// TIA Portal V19 export
FUNCTION_BLOCK "LAF_PlcDiag"   // FB22, LAD
TITLE = LAF_PlcDiag / SPS Geraete Status
AUTHOR : Siemens Digital Industries
FAMILY : LAF
VERSION : 1.2
// The block reads the identification and maintenance data (I&M data) as well as the network addresses from the PLC and provides the information in the screen “Settings – PLC identification“. The screen is accessible in the setting screen.  
// 
// **PLC Data types**  
// * LAF_typePlcDiag  
// 
// **WinCC Screen**  
// ![Image](LAF_PlcDiag/en/image1.PNG)  
// 
// ---
// 
// **Block call example**  
// ![Image](LAF_PlcDiag/en/image5.PNG)  
// 
// ---
// 
// **Calling interface**  
// The block will be called once only in the cyclic program. The call takes place in the software unit CentralFunctions -> 05_Diagnostics -> [CallDiagnostic](../Functions/CallDiagnostic.htm)  
// 
// **Internally used “Extended instructions / blocks“**  
// GET_IM_DATA, RDREC, S_CONV, MOVE_BLK_VARIANT  
// 
// **Parameters**  
// This block is provided with “pre-defined actual parameters” for structured data types, user constants, system constants etc. Therefor these parameters have to be modified only slightly or not at all, if the symbols of DBs, user constants, and system constants have not been changed.  
// In the case of LAF_PlcDiag you only have to write the correct information on the input parameter localProfinetInterface.
// 
// **Get parameter information:**..
// **localCommon**  
// ![Image](LAF_PlcDiag/en/image2.PNG)  
// 
// ---
// 
// **localProfinetInterface**  
// ![Image](LAF_PlcDiag/en/image3.PNG)
// Der Baustein liest die Identification und Maintenance Daten (I&M-Daten), sowie die Netzwerkadressen der CPU aus und stellt diese in dem Bild „SYSTEM_SETTINGS“ zur Verfügung. Das Bild ist erreichbar über den Button „System“ (aus jedem Bild, rechts unten).  
// 
// **PLC-Datentypen**  
//  LSicar_typePlcDiag  
//  
// **WinCC-Bild**  
// 
// ![Image](LSicar_typePlcDiag/de/image1.PNG)  
// 
// **Beispielaufruf**  
// Abbildung in Kontaktplan (KOP), ohne Parameterbeschaltung. D:\Software\Symbols_Icons\BMPs-JPGs-PNGs\Verschiedene\symb_user_goto_transparent.pngEin lauffähiger Programm-Aufruf hierzu ist im „SICAR-StartUp“-Projekt enthalten, incl. der notwendigen HMI-Variablen zur Darstellung der der Werte auf dem HMI.  
// 
// **Aufrufschnittstelle**  
// Der Baustein wird einmalig im zyklischen Programm aufgerufen.  
// 
// **Intern verwendete „Erweiterte Anweisungen / Bausteine“**  
// GET_IM_DATA, RDREC, S_CONV, MOVE_BLK_VARIANT 
// 
// **Parameter**  
// Der Baustein ist mit "Vordefinierten Aktualparametern" versehen für Strukturvariablen, Anwender- und Systemkonstanten etc., die dadurch nicht oder nur geringfügig angepasst werden müssen, vorausgesetzt die Symbolischen Namen von DBs, Anwender-/Systemkonstanten etc. wurden nicht geändert. Die Anpassungen sind notwendig beim Index [i], z.B. für den BA-Bereich oder die HMI-/Panelnummer.  
// * Der Index ist vorbesetzt mit dem Wert [0]. Damit wird auf den Index 0 (Dummy) verwiesen. Sofern der Baustein-Parameter nicht benötigt wird, sind keine Anpassungen notwendig, andernfalls muss der Indexwert angepasst werden. 
// oder  
// * Der Index ist vorbesetzt mit [???]. Dies führt dazu, dass der Aktualparameter beim Bausteinaufruf rot markiert wird; um darauf aufmerksam zu machen, dass der Indexwert des Aktualparameters angepasst werden muss!
// stored: Access Published, IsIECCheckEnabled true, MemoryReserve 100, SetENOAutomatically true
   VAR_INPUT
      localCommon { ExternalAccessible := 'False'; ExternalVisible := 'False'; ExternalWritable := 'False'} : HW_SUBMODULE;   // Systemkonstante: Local~PROFINET_IO-System / System constant: Local~Common
      localProfinetInterface { ExternalAccessible := 'False'; ExternalVisible := 'False'; ExternalWritable := 'False'} : HW_INTERFACE;   // Systemkonatante: Local~PROFINET-Interface_... / System constant: Local~PROFINET-Interface_...
      firstCycle { ExternalAccessible := 'False'; ExternalVisible := 'False'; ExternalWritable := 'False'} : Bool;   // SystemFlag: FirstCycle / System Flag: FirstCycle
   END_VAR
   VAR_IN_OUT
      diagDataHmi : "LAF_typePlcDiag";   // PLC-Diagnostic Data
   END_VAR
   VAR
      statLocalCommon { ExternalAccessible := 'False'; ExternalVisible := 'False'; ExternalWritable := 'False'} : HW_SUBMODULE;   // HW submodul
      statLocProfinetInterface { ExternalAccessible := 'False'; ExternalVisible := 'False'; ExternalWritable := 'False'} : HW_INTERFACE;   // HW interface
      instGetImData0 { ExternalAccessible := 'False'; ExternalVisible := 'False'; ExternalWritable := 'False'} : Get_IM_Data;   // I&M 0-Daten
      statGetImData0ErrorSaved { ExternalAccessible := 'False'; ExternalVisible := 'False'; ExternalWritable := 'False'} : Word;   // I&M 0-Daten
      instGetImData1 { ExternalAccessible := 'False'; ExternalVisible := 'False'; ExternalWritable := 'False'} : Get_IM_Data;   // I&M 1-Daten
      statGetImData1ErrorSaved { ExternalAccessible := 'False'; ExternalVisible := 'False'; ExternalWritable := 'False'} : Word;   // I&M 1-Daten
      instGetImData2 { ExternalAccessible := 'False'; ExternalVisible := 'False'; ExternalWritable := 'False'} : Get_IM_Data;   // I&M 2-Daten
      statGetImData2ErrorSaved { ExternalAccessible := 'False'; ExternalVisible := 'False'; ExternalWritable := 'False'} : Word;   // I&M 2-Daten
      instGetImData3 { ExternalAccessible := 'False'; ExternalVisible := 'False'; ExternalWritable := 'False'} : Get_IM_Data;   // I&M 3-Daten
      statGetImData3ErroSaved { ExternalAccessible := 'False'; ExternalVisible := 'False'; ExternalWritable := 'False'} : Word;   // I&M 3-Daten
      instReadRecord { ExternalAccessible := 'False'; ExternalVisible := 'False'; ExternalWritable := 'False'} : RDREC;   // RDREC
      statReadRecordResult { ExternalAccessible := 'False'; ExternalVisible := 'False'; ExternalWritable := 'False'} : Array[0..199] of Byte;   // RDREC-Record
      statStartNetAddresses { ExternalAccessible := 'False'; ExternalVisible := 'False'; ExternalWritable := 'False'} : USInt;   // Anfang der Netzadressesn (MAC, IP, Subnet, ...) / Start of net adresses (MAC, IP, Subnet, ...)
      statIm1PlDesiLocIdLen { ExternalAccessible := 'False'; ExternalVisible := 'False'; ExternalWritable := 'False'} : Int;   // Länge/Anzahl Zeichen von String "IuM_1_PlantDesign_LocIdent" / Lenght/Number of signs of string "IuM_1_PlantDesign_LocIdent"
      statRisEdgeReadAll { ExternalAccessible := 'False'; ExternalVisible := 'False'; ExternalWritable := 'False'} : Bool;   // Rising edge read all / Steigende Flanke read all
      statPosPulseReadAll { ExternalAccessible := 'False'; ExternalVisible := 'False'; ExternalWritable := 'False'} : Bool;   // Pos pulse read all / Pos. Impuls read all
      statErrorText { ExternalAccessible := 'False'; ExternalVisible := 'False'; ExternalWritable := 'False'} : String[#LENGTH_ERROR_TEXT] := STRING#'Error - Not readable data';   // Error text / Fehlertext
   END_VAR
   VAR_TEMP
      tempNetAddress : USInt;   // Netzadresse / Net address
      tempReadRecordResult6 : USInt;   // Type conversion / Typ Konvertierung
   END_VAR
   VAR CONSTANT
      VALUE_2 : USInt := 2;   // Konstante 2 / Const 2
      VALUE_4 : USInt := 4;   // 4Byte-1DW / 4 byte-1DW
      INDEX_ADDRESS_1ST_SIGN : USInt := 6;   // Indexadresse 1.Zeichen / Index address
      LENGTH_ERROR_TEXT : DInt := 30;   // Length error text / Zeichenlänge Fehlertext
   END_VAR
   VAR_TEMP   // added for the SCL form of the ladder/FBD networks
      _w1 : Bool;
   END_VAR
BEGIN

REGION Network 1: Header Info / Änderungshistorie
   // SIEMENS AG / (c)Copyright 2024
   // ------------------------------------------------------------------------------
   // Title:            LAF_InterfaceSignalsBool
   // Comment/Function: The block reads the identification and maintenance data (I&M data) as well as the network addresses from the PLC and provides the information in the screen “Settings – PLC identification“. 
   // Library/Family:  Library of Automation Framework
   // Author:               Siemens Digital Industry
   // Tested with:      S7-PLCSIM Advanced 6.0
   // Engineering:     TIA Portal V19
   // Restrictions:      ---
   // Requirements:  ---
   // ------------------------------------------------------------------------------
   // Change log table:
   // Version | Date | Expert in charge | Changes applied
   // -------|---------|-------------|--------------------------------------------
   // 01.02.00 | 30.09.2024 | SIMATIC Systems Support | First released version
   // Die Änderungshistorie wird nur in englischer Editiersprache geführt.
END_REGION

REGION Network 2: Description / Beschreibung
   // **Operation mode Automatic / Manual**  
   // The block is not assigned to any operation mode.  
   // 
   // **Alarms**  
   // The block does not generate alarms.  
   // 
   // #### PLC Data types 
   // * [LAF_typePlcDiag](../Library%20Types/LAF_typePlcDiag.htm)  
   // 
   // #### WinCC-Screen objects  
   // 
   // **WinCC Screen**  
   // The screen is located in the project in HMI part under “Screens” -> “11_Settings”.  
   // It consists of several WinCC objects and contains the shown below information.  
   // The Identification and Maintenance Data as well as the CPU net addresses are read once after a CPU warm start and displayed in the shown screen.  
   // ![Image](LAF_PlcDiag/en/image4.PNG)  
   // 
   // 
   // #### Further information 
   // 
   // #### Update info 
   // 
   // #### Further documentation
   // **Betriebsart Automatik / Hand**  
   // Der Baustein ist keiner Betriebsart / Betriebsartenbereich zugeordnet.  
   // 
   // **Alarme**  
   // Der Baustein generiert keine Alarme.  
   // 
   // #### PLC-Datentypen 
   // Der PLC-Datentyp „_typePlcDiag“ enthält alle Informationen, die in der Visualisierung angezeigt werden.  
   // 
   // #### WinCC-Bildobjekte 
   // **WinCC-Bild**  
   // Das Bild befindet sich im Projekt im HMI-Teil unter „Bilder“. Es ist erstellt aus mehreren einzelnen WinCC-Objekten und enthält die dargestellten Informationen.  
   // 
   // ![Image](LSicar_typePlcDiag/de/image2.PNG) 
   // 
   // 
   // #### Weitere Hinweise
   // 
   // #### Updateinfo 
   // 
   // #### Weitere Dokumente
END_REGION

REGION Network 3: Preset values after restart / Werte vorbesetzen nach Neustart
   // Initialization of the values / Initialisieren der  Werte
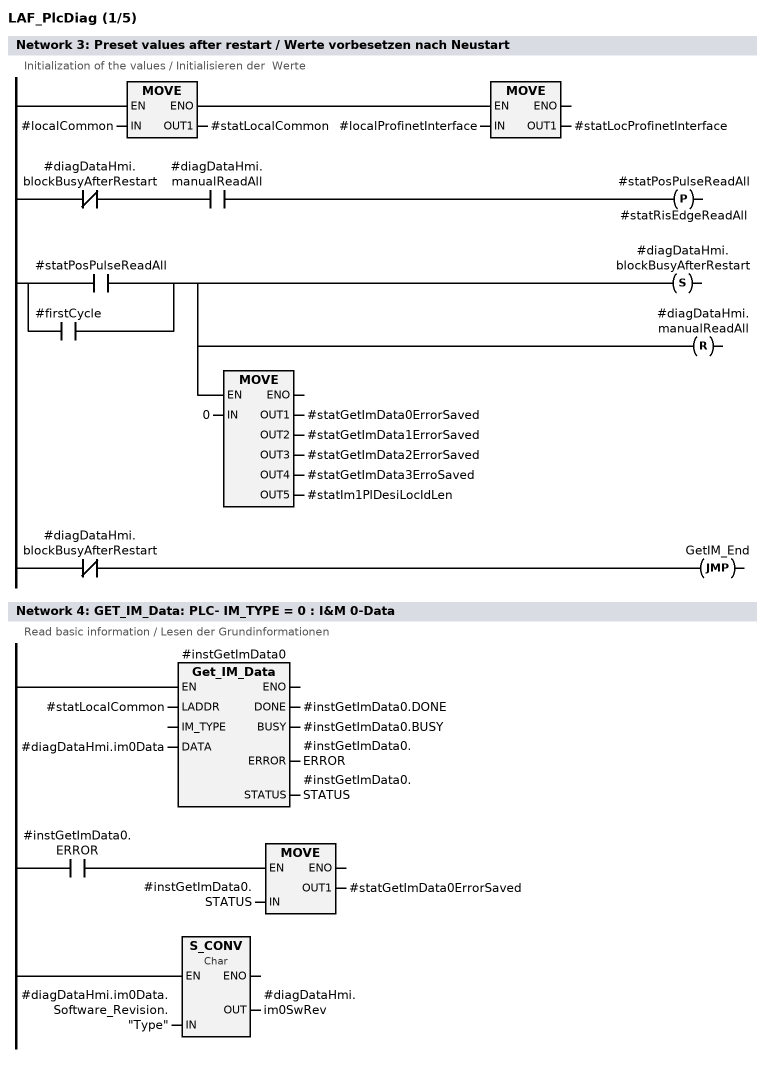
   #statLocalCommon := #localCommon;
   #statLocProfinetInterface := #localProfinetInterface;
   #_w1 := NOT #diagDataHmi.blockBusyAfterRestart AND #diagDataHmi.manualReadAll;
   #statPosPulseReadAll := #_w1 AND NOT #statRisEdgeReadAll;   // rising edge
   #statRisEdgeReadAll := #_w1;
   IF #statPosPulseReadAll OR #firstCycle THEN
       #diagDataHmi.blockBusyAfterRestart := TRUE;
       #diagDataHmi.manualReadAll := FALSE;
       #statGetImData0ErrorSaved := 0;
       #statGetImData1ErrorSaved := 0;
       #statGetImData2ErrorSaved := 0;
       #statGetImData3ErroSaved := 0;
       #statIm1PlDesiLocIdLen := 0;
   END_IF;
   IF NOT #diagDataHmi.blockBusyAfterRestart THEN GOTO GetIM_End; END_IF;
END_REGION

REGION Network 4: GET_IM_Data: PLC- IM_TYPE = 0 : I&M 0-Data
   // Read basic information / Lesen der Grundinformationen
   RUNG wire#powerrail
      #instGetImData0.Get_IM_Data(LADDR := #statLocalCommon, IM_TYPE :=, DATA := #diagDataHmi.im0Data, DONE => #instGetImData0.DONE, BUSY => #instGetImData0.BUSY, ERROR => #instGetImData0.ERROR, STATUS => #instGetImData0.STATUS)
   END_RUNG
   RUNG wire#powerrail
      Contact( #instGetImData0.ERROR )
      Move(in := #instGetImData0.STATUS, out1 => #statGetImData0ErrorSaved)
   END_RUNG
   RUNG wire#powerrail
      { S7_Templates := "[src_type := Char, dest_type := String]" } S_CONV(IN := #diagDataHmi.im0Data.Software_Revision."Type", OUT => #diagDataHmi.im0SwRev)
   END_RUNG
   // the same network as SCL:
   #instGetImData0(LADDR := #statLocalCommon,   // Get_IM_Data
                   DATA := #diagDataHmi.im0Data,
                   DONE => #instGetImData0.DONE,
                   BUSY => #instGetImData0.BUSY,
                   ERROR => #instGetImData0.ERROR,
                   STATUS => #instGetImData0.STATUS);
   IF #instGetImData0.ERROR THEN #statGetImData0ErrorSaved := #instGetImData0.STATUS; END_IF;
   S_CONV(IN := #diagDataHmi.im0Data.Software_Revision."Type", OUT => #diagDataHmi.im0SwRev);
END_REGION

REGION Network 5: GET_IM_Data: PLC- IM_TYPE = 11: I&M 1-Data
   // Read functional description an designation of the PLC / Lesen der Functionsbeschreibung und Bezeichnung der SPS
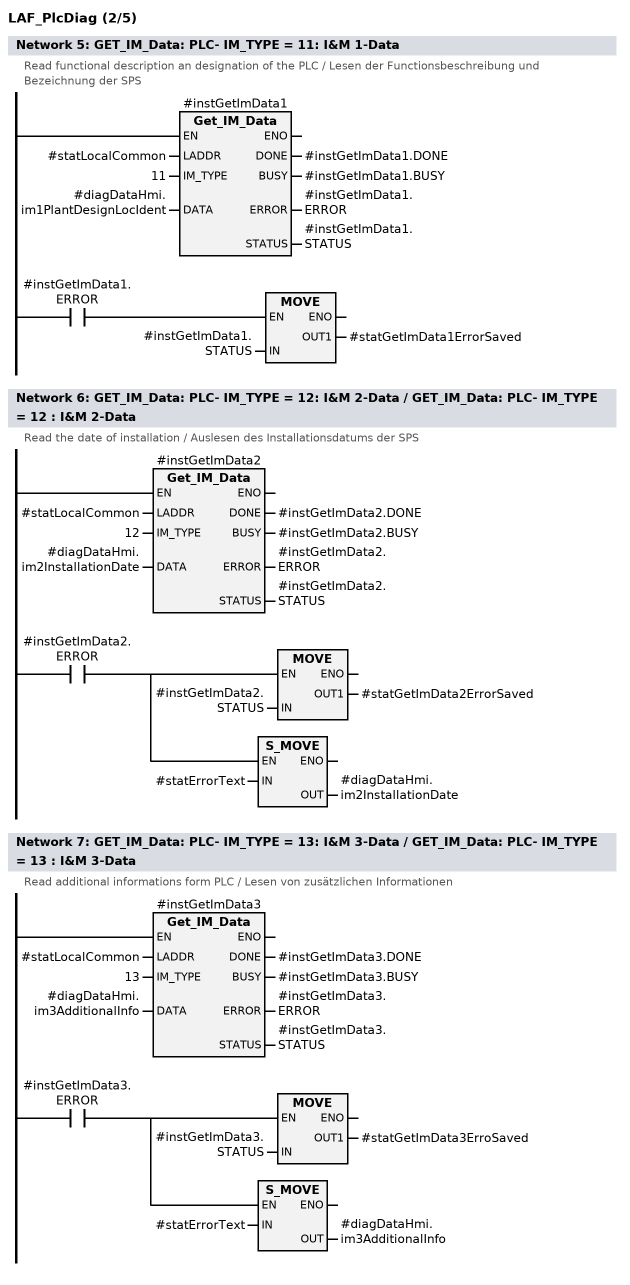
   RUNG wire#powerrail
      #instGetImData1.Get_IM_Data(LADDR := #statLocalCommon, IM_TYPE := 11, DATA := #diagDataHmi.im1PlantDesignLocIdent, DONE => #instGetImData1.DONE, BUSY => #instGetImData1.BUSY, ERROR => #instGetImData1.ERROR, STATUS => #instGetImData1.STATUS)
   END_RUNG
   RUNG wire#powerrail
      Contact( #instGetImData1.ERROR )
      Move(in := #instGetImData1.STATUS, out1 => #statGetImData1ErrorSaved)
   END_RUNG
   // the same network as SCL:
   #instGetImData1(LADDR := #statLocalCommon,   // Get_IM_Data
                   IM_TYPE := 11,
                   DATA := #diagDataHmi.im1PlantDesignLocIdent,
                   DONE => #instGetImData1.DONE,
                   BUSY => #instGetImData1.BUSY,
                   ERROR => #instGetImData1.ERROR,
                   STATUS => #instGetImData1.STATUS);
   IF #instGetImData1.ERROR THEN #statGetImData1ErrorSaved := #instGetImData1.STATUS; END_IF;
END_REGION

REGION Network 6: GET_IM_Data: PLC- IM_TYPE = 12: I&M 2-Data / GET_IM_Data: PLC- IM_TYPE = 12 : I&M 2-Data
   // Read the date of installation / Auslesen des Installationsdatums der SPS
   RUNG wire#powerrail
      #instGetImData2.Get_IM_Data(LADDR := #statLocalCommon, IM_TYPE := 12, DATA := #diagDataHmi.im2InstallationDate, DONE => #instGetImData2.DONE, BUSY => #instGetImData2.BUSY, ERROR => #instGetImData2.ERROR, STATUS => #instGetImData2.STATUS)
   END_RUNG
   RUNG wire#powerrail
      Contact( #instGetImData2.ERROR )
      wire#w1
      Move(in := #instGetImData2.STATUS, out1 => #statGetImData2ErrorSaved)
   END_RUNG
   RUNG wire#w1
      S_Move(in := #statErrorText, out => #diagDataHmi.im2InstallationDate)
   END_RUNG
   // the same network as SCL:
   #instGetImData2(LADDR := #statLocalCommon,   // Get_IM_Data
                   IM_TYPE := 12,
                   DATA := #diagDataHmi.im2InstallationDate,
                   DONE => #instGetImData2.DONE,
                   BUSY => #instGetImData2.BUSY,
                   ERROR => #instGetImData2.ERROR,
                   STATUS => #instGetImData2.STATUS);
   IF #instGetImData2.ERROR THEN
       #statGetImData2ErrorSaved := #instGetImData2.STATUS;
       #diagDataHmi.im2InstallationDate := #statErrorText;
   END_IF;
END_REGION

REGION Network 7: GET_IM_Data: PLC- IM_TYPE = 13: I&M 3-Data / GET_IM_Data: PLC- IM_TYPE = 13 : I&M 3-Data
   // Read additional informations form PLC / Lesen von zusätzlichen Informationen
   RUNG wire#powerrail
      #instGetImData3.Get_IM_Data(LADDR := #statLocalCommon, IM_TYPE := 13, DATA := #diagDataHmi.im3AdditionalInfo, DONE => #instGetImData3.DONE, BUSY => #instGetImData3.BUSY, ERROR => #instGetImData3.ERROR, STATUS => #instGetImData3.STATUS)
   END_RUNG
   RUNG wire#powerrail
      Contact( #instGetImData3.ERROR )
      wire#w1
      Move(in := #instGetImData3.STATUS, out1 => #statGetImData3ErroSaved)
   END_RUNG
   RUNG wire#w1
      S_Move(in := #statErrorText, out => #diagDataHmi.im3AdditionalInfo)
   END_RUNG
   // the same network as SCL:
   #instGetImData3(LADDR := #statLocalCommon,   // Get_IM_Data
                   IM_TYPE := 13,
                   DATA := #diagDataHmi.im3AdditionalInfo,
                   DONE => #instGetImData3.DONE,
                   BUSY => #instGetImData3.BUSY,
                   ERROR => #instGetImData3.ERROR,
                   STATUS => #instGetImData3.STATUS);
   IF #instGetImData3.ERROR THEN
       #statGetImData3ErroSaved := #instGetImData3.STATUS;
       #diagDataHmi.im3AdditionalInfo := #statErrorText;
   END_IF;
END_REGION

REGION Network 8: Read IP adress / Lesen der IP Adresse
   // Once only read RDREC (IP-Adresse): after PLC-restart or manual read from HMI / Einmaliges Lesen RDREC: nach SPS - Neustart oder manueller Anstoss vom HMI
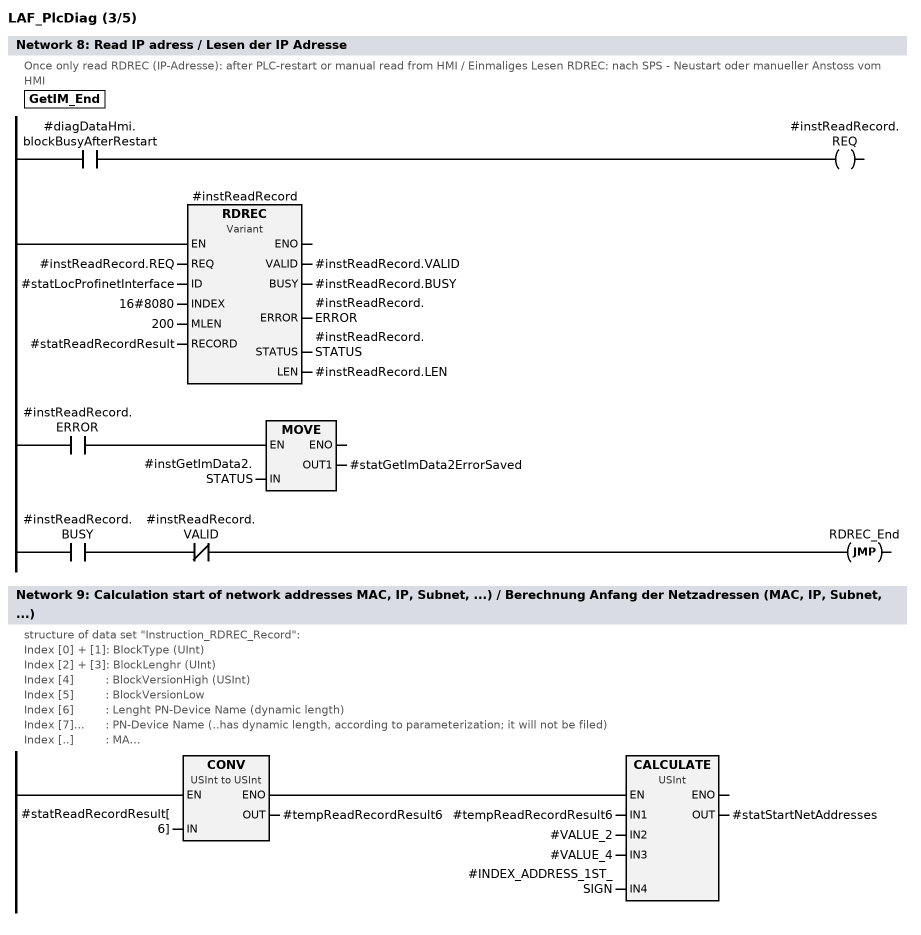
   Label( GetIM_End )
   RUNG wire#powerrail
      Contact( #diagDataHmi.blockBusyAfterRestart )
      Coil( #instReadRecord.REQ )
   END_RUNG
   RUNG wire#powerrail
      { S7_Templates := "[ptr_type := Variant, id_type := HW_IO, index_type := DInt, len_type := UInt]" } #instReadRecord.RDREC(REQ := #instReadRecord.REQ, ID := #statLocProfinetInterface, INDEX := 16#8080, MLEN := 200, RECORD := #statReadRecordResult, VALID => #instReadRecord.VALID, BUSY => #instReadRecord.BUSY, ERROR => #instReadRecord.ERROR, STATUS => #instReadRecord.STATUS, LEN => #instReadRecord.LEN)
   END_RUNG
   RUNG wire#powerrail
      Contact( #instReadRecord.ERROR )
      Move(in := #instGetImData2.STATUS, out1 => #statGetImData2ErrorSaved)
   END_RUNG
   RUNG wire#powerrail
      Contact( #instReadRecord.BUSY )
      I_Contact( #instReadRecord.VALID )
      JumpCoil( RDREC_End )
   END_RUNG
   // the same network as SCL:
   GetIM_End:
   #instReadRecord.REQ := #diagDataHmi.blockBusyAfterRestart;
   #instReadRecord(REQ := #instReadRecord.REQ,   // RDREC
                   ID := #statLocProfinetInterface,
                   INDEX := 16#8080,
                   MLEN := 200,
                   RECORD := #statReadRecordResult,
                   VALID => #instReadRecord.VALID,
                   BUSY => #instReadRecord.BUSY,
                   ERROR => #instReadRecord.ERROR,
                   STATUS => #instReadRecord.STATUS,
                   LEN => #instReadRecord.LEN);
   IF #instReadRecord.ERROR THEN #statGetImData2ErrorSaved := #instGetImData2.STATUS; END_IF;
   IF #instReadRecord.BUSY AND NOT #instReadRecord.VALID THEN GOTO RDREC_End; END_IF;
END_REGION

REGION Network 9: Calculation start of network addresses MAC, IP, Subnet, ...) / Berechnung Anfang der Netzadressen (MAC, IP, Subnet, ...)
   // structure of data set "Instruction_RDREC_Record":
   // Index [0] + [1]: BlockType (UInt)
   // Index [2] + [3]: BlockLenghr (UInt)
   // Index [4]         : BlockVersionHigh (USInt)
   // Index [5]         : BlockVersionLow
   // Index [6]         : Lenght PN-Device Name (dynamic length)
   // Index [7]...      : PN-Device Name (..has dynamic length, according to parameterization; it will not be filed)
   // Index [..]         : MAC
   // Index [..]         : IP
   // Index [..]         : SubnetMask
   // Index [..]         : Standard Gateway (is not filed)
   // Aufbau des Datensatzes "Instruction_RDREC_Record":
   // Index [0] + [1]: BlockType (UInt)
   // Index [2] + [3]: BlockLenghr (UInt)
   // Index [4]         : BlockVersionHigh (USInt)
   // Index [5]         : BlockVersionLow
   // Index [6]         : Lenght PN-Device Name (dynamische Länge)
   // Index [7]...      : PN-Device Name (..hat dynamische Länge, je nach Parametrierung; wird nicht abgelegt)
   // Index [..]         : MAC
   // Index [..]         : IP
   // Index [..]         . SubnetMask
   // Index [..]         : Standard Gateway (wird nicht abgelegt)
   RUNG wire#powerrail
      { S7_Templates := "[SrcType := USInt, DestType := USInt]" } Convert(in := #statReadRecordResult[6], out => #tempReadRecordResult6)
      { S7_Templates := "SrcType := USInt"; S7_Expression := "IN3 - ((IN1 + IN2) MOD IN3) + IN1 + IN4" } Calculate(in1 := #tempReadRecordResult6, in2 := #VALUE_2, in3 := #VALUE_4, in4 := #INDEX_ADDRESS_1ST_SIGN, out => #statStartNetAddresses)
   END_RUNG
   // the same network as SCL:
   #tempReadRecordResult6 := USINT_TO_USINT(#statReadRecordResult[6]);
   #statStartNetAddresses := #VALUE_4 - ((#tempReadRecordResult6 + #VALUE_2) MOD #VALUE_4) + #tempReadRecordResult6 + #INDEX_ADDRESS_1ST_SIGN;
END_REGION

REGION Network 10: Data routing into PLC_Data.Global MAC-Adresse / Daten Rangierung nach PLC_Data.Global MAC-Adresse
   // Copy the MAC adress to InOut variable / Kopieren der MAC Adresse an einer InOut Variable
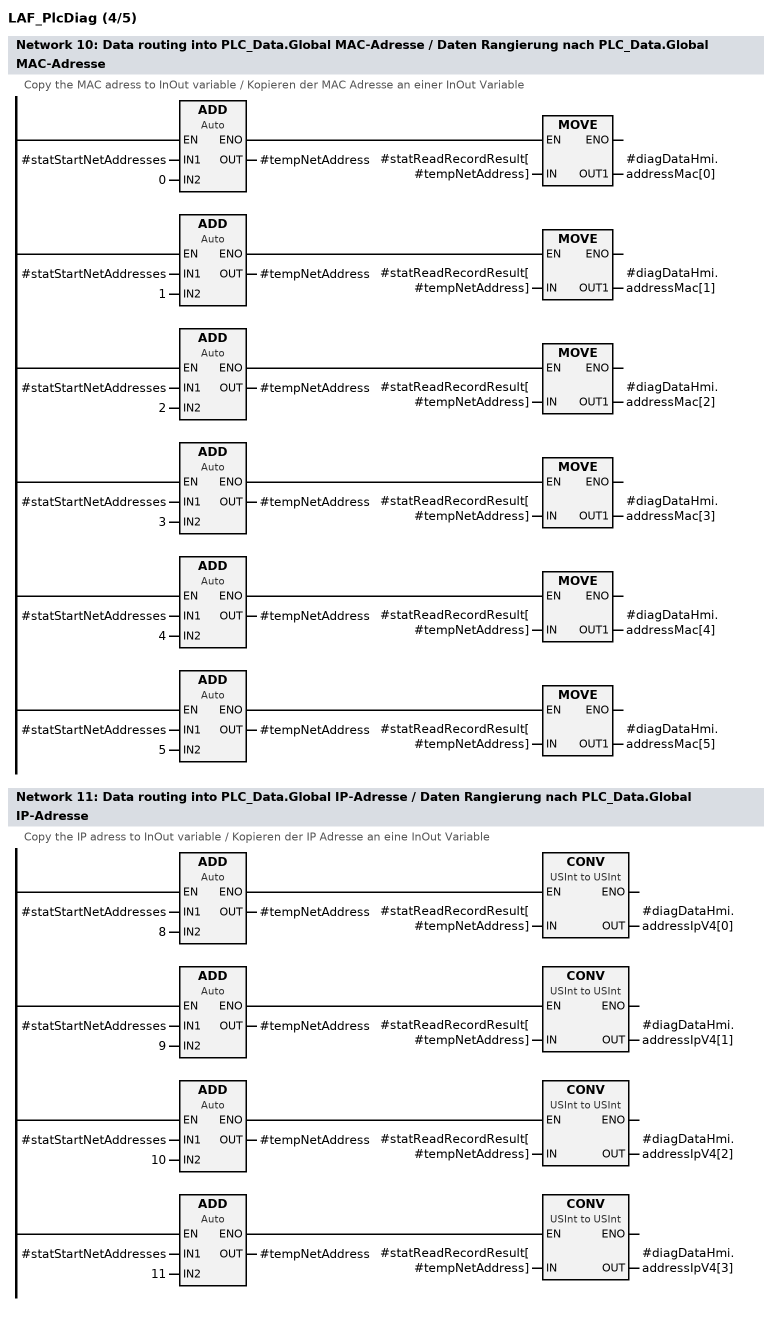
   RUNG wire#powerrail
      Add(in1 := #statStartNetAddresses, in2 := 0, out => #tempNetAddress)
      Move(in := #statReadRecordResult[#tempNetAddress], out1 => #diagDataHmi.addressMac[0])
   END_RUNG
   RUNG wire#powerrail
      Add(in1 := #statStartNetAddresses, in2 := 1, out => #tempNetAddress)
      Move(in := #statReadRecordResult[#tempNetAddress], out1 => #diagDataHmi.addressMac[1])
   END_RUNG
   RUNG wire#powerrail
      Add(in1 := #statStartNetAddresses, in2 := 2, out => #tempNetAddress)
      Move(in := #statReadRecordResult[#tempNetAddress], out1 => #diagDataHmi.addressMac[2])
   END_RUNG
   RUNG wire#powerrail
      Add(in1 := #statStartNetAddresses, in2 := 3, out => #tempNetAddress)
      Move(in := #statReadRecordResult[#tempNetAddress], out1 => #diagDataHmi.addressMac[3])
   END_RUNG
   RUNG wire#powerrail
      Add(in1 := #statStartNetAddresses, in2 := 4, out => #tempNetAddress)
      Move(in := #statReadRecordResult[#tempNetAddress], out1 => #diagDataHmi.addressMac[4])
   END_RUNG
   RUNG wire#powerrail
      Add(in1 := #statStartNetAddresses, in2 := 5, out => #tempNetAddress)
      Move(in := #statReadRecordResult[#tempNetAddress], out1 => #diagDataHmi.addressMac[5])
   END_RUNG
   // the same network as SCL:
   #tempNetAddress := #statStartNetAddresses + 0;
   #diagDataHmi.addressMac[0] := #statReadRecordResult[#tempNetAddress];
   #tempNetAddress := #statStartNetAddresses + 1;
   #diagDataHmi.addressMac[1] := #statReadRecordResult[#tempNetAddress];
   #tempNetAddress := #statStartNetAddresses + 2;
   #diagDataHmi.addressMac[2] := #statReadRecordResult[#tempNetAddress];
   #tempNetAddress := #statStartNetAddresses + 3;
   #diagDataHmi.addressMac[3] := #statReadRecordResult[#tempNetAddress];
   #tempNetAddress := #statStartNetAddresses + 4;
   #diagDataHmi.addressMac[4] := #statReadRecordResult[#tempNetAddress];
   #tempNetAddress := #statStartNetAddresses + 5;
   #diagDataHmi.addressMac[5] := #statReadRecordResult[#tempNetAddress];
END_REGION

REGION Network 11: Data routing into PLC_Data.Global IP-Adresse / Daten Rangierung nach PLC_Data.Global IP-Adresse
   // Copy the IP adress to InOut variable / Kopieren der IP Adresse an eine InOut Variable
   RUNG wire#powerrail
      Add(in1 := #statStartNetAddresses, in2 := 8, out => #tempNetAddress)
      { S7_Templates := "[SrcType := USInt, DestType := USInt]" } Convert(in := #statReadRecordResult[#tempNetAddress], out => #diagDataHmi.addressIpV4[0])
   END_RUNG
   RUNG wire#powerrail
      Add(in1 := #statStartNetAddresses, in2 := 9, out => #tempNetAddress)
      { S7_Templates := "[SrcType := USInt, DestType := USInt]" } Convert(in := #statReadRecordResult[#tempNetAddress], out => #diagDataHmi.addressIpV4[1])
   END_RUNG
   RUNG wire#powerrail
      Add(in1 := #statStartNetAddresses, in2 := 10, out => #tempNetAddress)
      { S7_Templates := "[SrcType := USInt, DestType := USInt]" } Convert(in := #statReadRecordResult[#tempNetAddress], out => #diagDataHmi.addressIpV4[2])
   END_RUNG
   RUNG wire#powerrail
      Add(in1 := #statStartNetAddresses, in2 := 11, out => #tempNetAddress)
      { S7_Templates := "[SrcType := USInt, DestType := USInt]" } Convert(in := #statReadRecordResult[#tempNetAddress], out => #diagDataHmi.addressIpV4[3])
   END_RUNG
   // the same network as SCL:
   #tempNetAddress := #statStartNetAddresses + 8;
   #diagDataHmi.addressIpV4[0] := USINT_TO_USINT(#statReadRecordResult[#tempNetAddress]);
   #tempNetAddress := #statStartNetAddresses + 9;
   #diagDataHmi.addressIpV4[1] := USINT_TO_USINT(#statReadRecordResult[#tempNetAddress]);
   #tempNetAddress := #statStartNetAddresses + 10;
   #diagDataHmi.addressIpV4[2] := USINT_TO_USINT(#statReadRecordResult[#tempNetAddress]);
   #tempNetAddress := #statStartNetAddresses + 11;
   #diagDataHmi.addressIpV4[3] := USINT_TO_USINT(#statReadRecordResult[#tempNetAddress]);
END_REGION

REGION Network 12: Data routing into PLC_Data.Global Subnet-Adresse / Daten Rangierung nach PLC_Data.Global Subnet-Adresse
   // Copy the subnet mask to InOut variable / Kopieren der Subnetz-Maske an eine InOut Variable
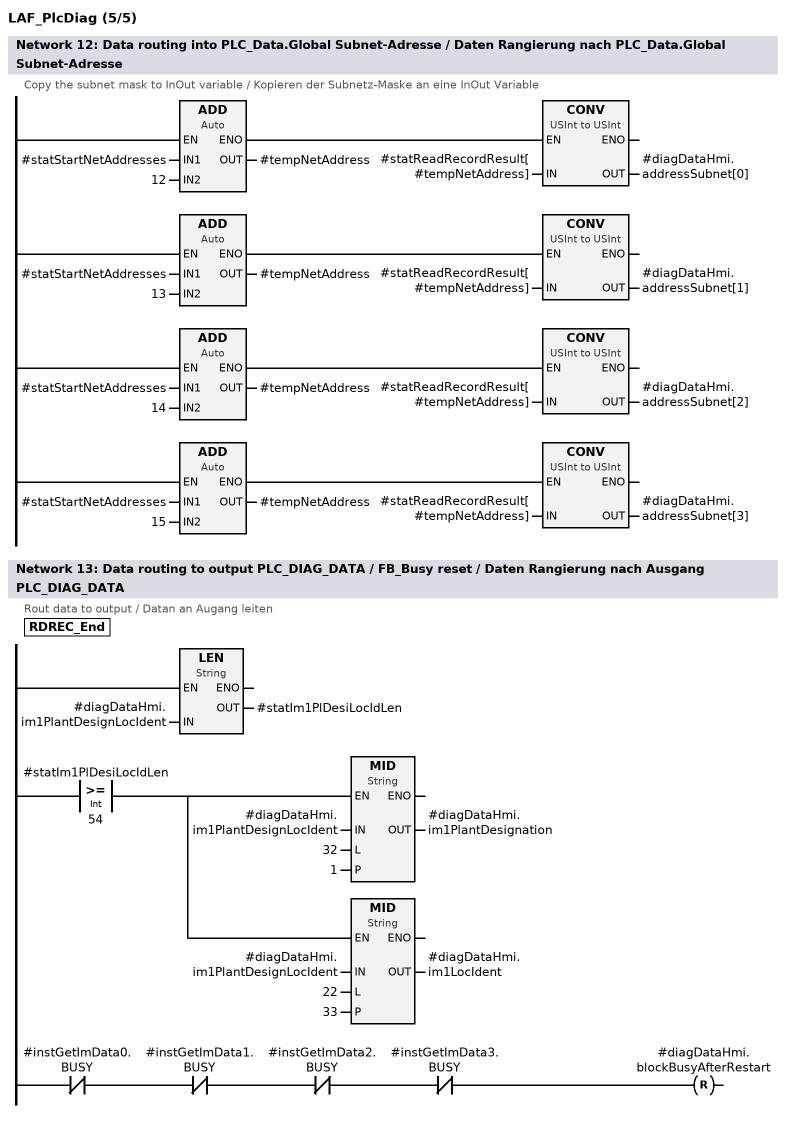
   RUNG wire#powerrail
      Add(in1 := #statStartNetAddresses, in2 := 12, out => #tempNetAddress)
      { S7_Templates := "[SrcType := USInt, DestType := USInt]" } Convert(in := #statReadRecordResult[#tempNetAddress], out => #diagDataHmi.addressSubnet[0])
   END_RUNG
   RUNG wire#powerrail
      Add(in1 := #statStartNetAddresses, in2 := 13, out => #tempNetAddress)
      { S7_Templates := "[SrcType := USInt, DestType := USInt]" } Convert(in := #statReadRecordResult[#tempNetAddress], out => #diagDataHmi.addressSubnet[1])
   END_RUNG
   RUNG wire#powerrail
      Add(in1 := #statStartNetAddresses, in2 := 14, out => #tempNetAddress)
      { S7_Templates := "[SrcType := USInt, DestType := USInt]" } Convert(in := #statReadRecordResult[#tempNetAddress], out => #diagDataHmi.addressSubnet[2])
   END_RUNG
   RUNG wire#powerrail
      Add(in1 := #statStartNetAddresses, in2 := 15, out => #tempNetAddress)
      { S7_Templates := "[SrcType := USInt, DestType := USInt]" } Convert(in := #statReadRecordResult[#tempNetAddress], out => #diagDataHmi.addressSubnet[3])
   END_RUNG
   // the same network as SCL:
   #tempNetAddress := #statStartNetAddresses + 12;
   #diagDataHmi.addressSubnet[0] := USINT_TO_USINT(#statReadRecordResult[#tempNetAddress]);
   #tempNetAddress := #statStartNetAddresses + 13;
   #diagDataHmi.addressSubnet[1] := USINT_TO_USINT(#statReadRecordResult[#tempNetAddress]);
   #tempNetAddress := #statStartNetAddresses + 14;
   #diagDataHmi.addressSubnet[2] := USINT_TO_USINT(#statReadRecordResult[#tempNetAddress]);
   #tempNetAddress := #statStartNetAddresses + 15;
   #diagDataHmi.addressSubnet[3] := USINT_TO_USINT(#statReadRecordResult[#tempNetAddress]);
END_REGION

REGION Network 13: Data routing to output PLC_DIAG_DATA / FB_Busy reset / Daten Rangierung nach Ausgang PLC_DIAG_DATA
   // Rout data to output / Datan an Augang leiten
   Label( RDREC_End )
   RUNG wire#powerrail
      { S7_Templates := "[str_type := String, return_type := Int]" } LEN(IN := #diagDataHmi.im1PlantDesignLocIdent, OUT => #statIm1PlDesiLocIdLen)
   END_RUNG
   RUNG wire#powerrail
      { S7_Templates := "SrcType := Int" } GE_Contact(in1 := #statIm1PlDesiLocIdLen, in2 := 54)
      wire#w1
      { S7_Templates := "value_type := String" } MID(IN := #diagDataHmi.im1PlantDesignLocIdent, L := 32, P := 1, OUT => #diagDataHmi.im1PlantDesignation)
   END_RUNG
   RUNG wire#w1
      { S7_Templates := "value_type := String" } MID(IN := #diagDataHmi.im1PlantDesignLocIdent, L := 22, P := 33, OUT => #diagDataHmi.im1LocIdent)
   END_RUNG
   RUNG wire#powerrail
      I_Contact( #instGetImData0.BUSY )
      I_Contact( #instGetImData1.BUSY )
      I_Contact( #instGetImData2.BUSY )
      I_Contact( #instGetImData3.BUSY )
      R_Coil( #diagDataHmi.blockBusyAfterRestart )
   END_RUNG
   // the same network as SCL:
   RDREC_End:
   LEN(IN := #diagDataHmi.im1PlantDesignLocIdent, OUT => #statIm1PlDesiLocIdLen);
   IF #statIm1PlDesiLocIdLen >= 54 THEN
       MID(IN := #diagDataHmi.im1PlantDesignLocIdent, L := 32, P := 1, OUT => #diagDataHmi.im1PlantDesignation);
       MID(IN := #diagDataHmi.im1PlantDesignLocIdent, L := 22, P := 33, OUT => #diagDataHmi.im1LocIdent);
   END_IF;
   IF NOT #instGetImData0.BUSY AND NOT #instGetImData1.BUSY AND NOT #instGetImData2.BUSY AND NOT #instGetImData3.BUSY THEN
       #diagDataHmi.blockBusyAfterRestart := FALSE;
   END_IF;
END_REGION
END_FUNCTION_BLOCK
